% RSLogix 500 project I2P JOB 9_RUSSELL_BAK008.RSS, saved by version 10.00.00.00 %
PROJECT "ML02A"    % processor: Bul.1763 MicroLogix 1100 Series B %

PROGRAM FILES
  LAD 2   4 rungs

DATA FILES
  O0 OUTPUT  4 elements
  I1 INPUT  6 elements
  S2 STATUS  66 elements
  B3 BINARY  1 elements
  T4 TIMER  1 elements
  C5 COUNTER  1 elements
  R6 CONTROL  1 elements
  N7 INTEGER  1 elements
  F8 FLOAT  1 elements

LADDER 2
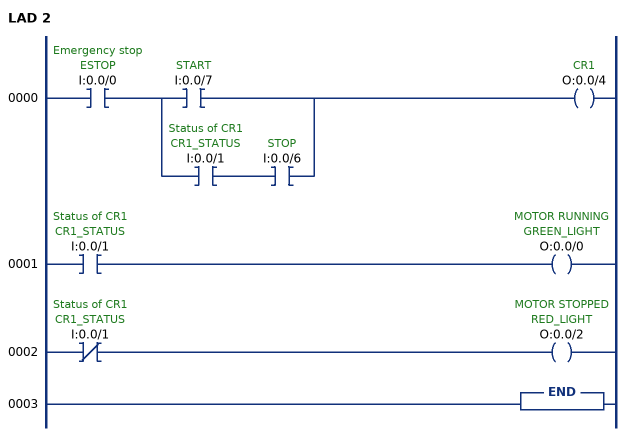
% Rung: 0 %  % edit flag set %
SOR XIC I:0.0/0 BST XIC I:0.0/7 NXB XIC I:0.0/1 XIC I:0.0/6 BND OTE O:0.0/4 EOR
%   I:0.0/0  ESTOP  "Emergency stop" %
%   I:0.0/7  "START" %
%   I:0.0/1  CR1_STATUS  "Status of CR1" %
%   I:0.0/6  "STOP" %
%   O:0.0/4  CR1 %
% Rung: 1 %  % edit flag set %
SOR XIC I:0.0/1 OTE O:0.0/0 EOR
%   I:0.0/1  CR1_STATUS  "Status of CR1" %
%   O:0.0/0  GREEN_LIGHT  "MOTOR RUNNING" %
% Rung: 2 %  % edit flag set %
SOR XIO I:0.0/1 OTE O:0.0/2 EOR
%   I:0.0/1  CR1_STATUS  "Status of CR1" %
%   O:0.0/2  RED_LIGHT  "MOTOR STOPPED" %
% Rung: 3 %
SOR END EOR

OTHER DOCUMENTED ADDRESSES
  I:0.0/2  CR2_STATUS  "Status of control relay 2"
  I:0.0/3  3PSS_A  "3 position selector switch A position"
  I:0.0/4  3PSS_B  "3 position selector switch B position"
  I:0.0/5  2PSS  "2 position selector switch"
  I:0.0/8  PB3  "Normally open pushbutton"
  O:0.0/1  YELLOW_LIGHT  "Yellow light"
  O:0.0/3  BLUE_LIGHT  "Blue light"
  O:0.0/5  CR2  "Contro relay 2"
